FUNCTION_BLOCK WRITE_MQTT_FIXED
  {SET_ATTRIBUTE(OpcUa, SERVICE)}
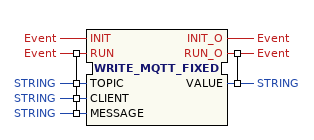
  EVENT_INPUT
    INIT;
    RUN WITH TOPIC, CLIENT, MESSAGE;
  END_EVENT
  EVENT_OUTPUT
    INIT_O;
    RUN_O WITH VALUE;
  END_EVENT
  VAR_INPUT
    TOPIC : STRING; {SET_ATTRIBUTE(OpcUa, Constant)}
    CLIENT : STRING; {SET_ATTRIBUTE(OpcUa, Variable)}
    MESSAGE : STRING; {SET_ATTRIBUTE(OpcUa, Constant)}
  END_VAR
  VAR_OUTPUT
    VALUE : STRING; {SET_ATTRIBUTE(OpcUa, Variable)}
  END_VAR
END_FUNCTION_BLOCK
